{attribute addProperty BoxType "EK1122-0000-0018"}
{attribute addProperty Id "Beckhoff_EP1xxxsub_EK1100EK1100_179A0949162A_0001_EP1008_0001_0016EP1008_772BB4148210.25A_0002_EP1008_0001_0017EP1008_772BB4148210.25A_0003_EP1008_0001_0018EP1008_772BB4148210.25A_0004_EP1008_0002_0016EP1008_772BB4148210.25A_0005_EP1008_0002_0017EP1008_772BB4148210.25A_0006_EP1008_0002_0018EP1008_772BB4148210.25A_0007_EP1008_0022_0016EP1008_772BB4148210.25A_0008_EP1008_0022_0017EP1008_772BB4148210.25A_0009_EP1018_0001_0016EP1018_772BB4148210.25A_0010_EP1018_0001_0017EP1018_772BB4148210.25A_0011_EP1018_0001_0018EP1018_772BB4148210.25A_0012_EP1018_0401_0016EP1018_772BB4148210.25A_0013_EP1018_0002_0016EP1018_772BB4148210.25A_0014_EP1018_0002_0017EP1018_772BB4148210.25A_0015_EP1018_0002_0018EP1018_772BB4148210.25A_0016_EP1098_0001_0016EP1098_772BB4148210.25A_0017_EP1098_0001_0017EP1098_772BB4148210.25A_0018_EP1111_0000_0016EP1111_0792AF759812.25A_0019_EP1111_0000_0017EP1111_0792AF759812.25A_0020_EP1111_0000_0018EP1111_0792AF759812.25A_0021_EP1111_0000_0019EP1111_0792AF759812.25A_0022_EP1111_0000_0020EP1111_0792AF759812.25A_0023_EP1111_0000_0021EP1111_0792AF759812.25A_0024_EP1122_0001_0016A_0024_EP1122_0001_0016_1C40CD3A1014268719478003.75"}
{attribute addProperty CRC "3081897315"}
{attribute addProperty SizeInBites "12140"}
{attribute addProperty SizeInBytes "68719478253.5"}
TYPE Beckhoff_EP1xxxEK1122_B7B20563 EXTENDS EK1122_179A0949 :
STRUCT
	{attribute addProperty Name "Beckhoff_EP1xxxsub_EK1100"}
	Beckhoff_EP1xxxsub_EK1100 : EK1100_179A0949;
	{attribute addProperty Name "A_0001_EP1008_0001_0016"}
	A_0001_EP1008_0001_0016 : EP1008_772BB414;
	{attribute addProperty Name "A_0002_EP1008_0001_0017"}
	A_0002_EP1008_0001_0017 : EP1008_772BB414;
	{attribute addProperty Name "A_0003_EP1008_0001_0018"}
	A_0003_EP1008_0001_0018 : EP1008_772BB414;
	{attribute addProperty Name "A_0004_EP1008_0002_0016"}
	A_0004_EP1008_0002_0016 : EP1008_772BB414;
	{attribute addProperty Name "A_0005_EP1008_0002_0017"}
	A_0005_EP1008_0002_0017 : EP1008_772BB414;
	{attribute addProperty Name "A_0006_EP1008_0002_0018"}
	A_0006_EP1008_0002_0018 : EP1008_772BB414;
	{attribute addProperty Name "A_0007_EP1008_0022_0016"}
	A_0007_EP1008_0022_0016 : EP1008_772BB414;
	{attribute addProperty Name "A_0008_EP1008_0022_0017"}
	A_0008_EP1008_0022_0017 : EP1008_772BB414;
	{attribute addProperty Name "A_0009_EP1018_0001_0016"}
	A_0009_EP1018_0001_0016 : EP1018_772BB414;
	{attribute addProperty Name "A_0010_EP1018_0001_0017"}
	A_0010_EP1018_0001_0017 : EP1018_772BB414;
	{attribute addProperty Name "A_0011_EP1018_0001_0018"}
	A_0011_EP1018_0001_0018 : EP1018_772BB414;
	{attribute addProperty Name "A_0012_EP1018_0401_0016"}
	A_0012_EP1018_0401_0016 : EP1018_772BB414;
	{attribute addProperty Name "A_0013_EP1018_0002_0016"}
	A_0013_EP1018_0002_0016 : EP1018_772BB414;
	{attribute addProperty Name "A_0014_EP1018_0002_0017"}
	A_0014_EP1018_0002_0017 : EP1018_772BB414;
	{attribute addProperty Name "A_0015_EP1018_0002_0018"}
	A_0015_EP1018_0002_0018 : EP1018_772BB414;
	{attribute addProperty Name "A_0016_EP1098_0001_0016"}
	A_0016_EP1098_0001_0016 : EP1098_772BB414;
	{attribute addProperty Name "A_0017_EP1098_0001_0017"}
	A_0017_EP1098_0001_0017 : EP1098_772BB414;
	{attribute addProperty Name "A_0018_EP1111_0000_0016"}
	A_0018_EP1111_0000_0016 : EP1111_0792AF75;
	{attribute addProperty Name "A_0019_EP1111_0000_0017"}
	A_0019_EP1111_0000_0017 : EP1111_0792AF75;
	{attribute addProperty Name "A_0020_EP1111_0000_0018"}
	A_0020_EP1111_0000_0018 : EP1111_0792AF75;
	{attribute addProperty Name "A_0021_EP1111_0000_0019"}
	A_0021_EP1111_0000_0019 : EP1111_0792AF75;
	{attribute addProperty Name "A_0022_EP1111_0000_0020"}
	A_0022_EP1111_0000_0020 : EP1111_0792AF75;
	{attribute addProperty Name "A_0023_EP1111_0000_0021"}
	A_0023_EP1111_0000_0021 : EP1111_0792AF75;
	{attribute addProperty Name "A_0024_EP1122_0001_0016"}
	A_0024_EP1122_0001_0016 : A_0024_EP1122_0001_0016_1C40CD3A;
END_STRUCT
END_TYPE

(* stored: Version 1.2.0.0, ProductVersion 3.1.4024.9
   DUT Beckhoff_EP1xxxEK1122_B7B20563: Id {f8ae042f-754d-4609-b6e5-69d6092cd303} *)
